Staubli VAL3: recvMsgBody.pgx

public program recvMsgBody()
  local bool l_bFlag
begin
  l_bFlag=false

  switch rosGenericMsg.header.nMsgType
    case 11
      call recvTrajPt(l_bFlag)
    break
    case 14
      call recvTrajPtFull(l_bFlag)
    break
    default
    break
  endSwitch

  if (l_bFlag)
    // move on to state 3: decode msg body
    nDataInState=3
  else
    // error whilst receiving msg body, reset state machine
    nDataInState=0
  endIf
end
